(* PLC project v0.6.04_CycleSemiAuto.project, CODESYS CODESYS V3.5 SP19 Patch 1 *)
(* stored: creationDateTime 2026-08-11T14:02:33.671560, modificationDateTime 2026-08-11T14:02:33.671560 *)

TYPE ST_Chain_Translation_Safety : STRUCT
  Idx301_EmergencyChainClosed : BOOL;  (* 1 = Boucle Urgence OK | 0 = Arrêt d'Urgence Appuyé 🔴 *)
  Idx302_SafeStopActive : BOOL;  (* 0 = Sain (Autorisé) | 1 = Arrêt Rapide Translation 🔴 *)
  Idx303_PowerCutOffActive : BOOL;  (* 0 = Puissance OK | 1 = Coupure Puissance 🔴 *)
  Idx304_LimitSwitchFwdActive : BOOL;  (* 0 = Sain | 1 = Fin de Course Extrême Avance 🔴 *)
  Idx305_LimitSwitchRevActive : BOOL;  (* 0 = Sain | 1 = Fin de Course Extrême Recul 🔴 *)
  Idx306_BypassLimitSwitch : BOOL;  (* 0 = Fins de course actives | 1 = Shuntés IHM ⚠️ *)
  Idx307_PositionDecoderIncoherent : BOOL;  (* 0 = Décodage 5 Capteurs OK | 1 = Incohérence Position 🔴 *)
  Idx308_HeightInterlockBlocking : BOOL;  (* 🆕 2026-08-06 : 0 = M1 ET M2 ≥ hauteur mini (ou bypass) | 1 = Translation bloquée (risque collision) 🔴 *)
END_STRUCT;
END_TYPE
